TYPE "UDT_ZC_RECETA_CIP_HOMOG"
VERSION : 0.1
   STRUCT
      TiempoAgitadorOn : Int;
      TiempoAgitadorOff : Int;
      TipoAgitacionVelocidad : Int := 0;
      VelocidadFijaAgitador : Real := 0.0;
      VolumenMinControlAgitador : Real := 0.0;
      VolumenMaxControlAgitador : Real := 0.0;
      VelocidadMinAgitador : Real := 0.0;
      VelocidadMaxAgitador : Real := 0.0;
      SPTemperatura : Real;
      HisteresisTemp : Real;
   END_STRUCT;

END_TYPE

